{attribute 'GeneratedUsingTerminal: EL3122--0000'}
{attribute addProperty BoxType "EL3122--0000"}
{attribute addProperty Id "Channel_1AT %I*Channel_7539AA333Channel_2AT %I*Channel_7539AA333WcStateAT %I*WcState_9091E0EB2InfoDataAT %I*InfoData_94A18F5E2"}
{attribute addProperty CRC "1578362931"}
{attribute addProperty Size "10"}
TYPE EL3122_5E13E833 EXTENDS EtcSlaveTerminalBase_947E5A46 :
STRUCT
	{attribute addProperty Name "Channel_1"}
	Channel_1 : Channel_7539AA33;
	{attribute addProperty Name "Channel_2"}
	Channel_2 : Channel_7539AA33;
	{attribute addProperty Name "WcState"}
	WcState : WcState_9091E0EB;
	{attribute addProperty Name "InfoData"}
	InfoData : InfoData_94A18F5E;
END_STRUCT
END_TYPE

(* stored: Version 1.2.0.0, ProductVersion 3.1.4024.9
   DUT EL3122_5E13E833: Id {f50a425e-3ea8-4c3c-8036-ebcc623b8780} *)
